// TIA Portal V20 export
FUNCTION "PLC数据交换" : Void   // FC1, LAD
{ S7_Optimized_Access := 'TRUE' }
// stored: SetENOAutomatically false
BEGIN

REGION Network 1
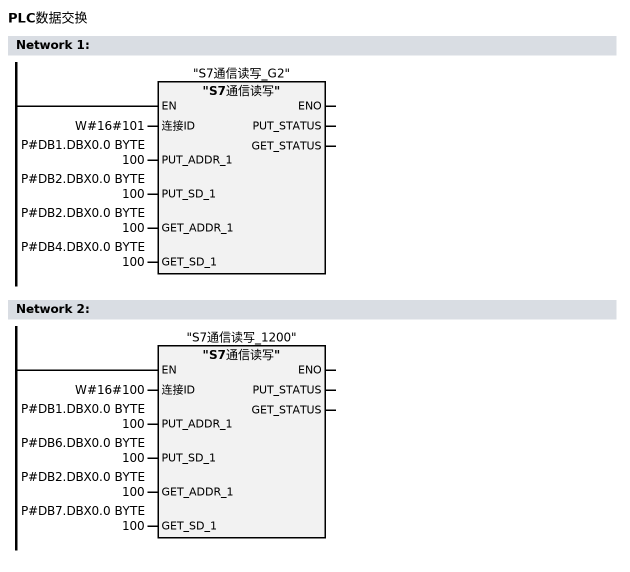
   RUNG wire#powerrail
      "S7通信读写_G2"(连接ID := W#16#101, PUT_ADDR_1 := P#DB1.DBX0.0 BYTE 100, PUT_SD_1 := P#DB2.DBX0.0 BYTE 100, GET_ADDR_1 := P#DB2.DBX0.0 BYTE 100, GET_SD_1 := P#DB4.DBX0.0 BYTE 100, PUT_STATUS =>, GET_STATUS =>)
   END_RUNG
   // the same network as SCL:
   "S7通信读写_G2"(连接ID := W#16#101,   // "S7通信读写"
               PUT_ADDR_1 := P#DB1.DBX0.0 BYTE 100,
               PUT_SD_1 := P#DB2.DBX0.0 BYTE 100,
               GET_ADDR_1 := P#DB2.DBX0.0 BYTE 100,
               GET_SD_1 := P#DB4.DBX0.0 BYTE 100);
END_REGION

REGION Network 2
   RUNG wire#powerrail
      "S7通信读写_1200"(连接ID := W#16#100, PUT_ADDR_1 := P#DB1.DBX0.0 BYTE 100, PUT_SD_1 := P#DB6.DBX0.0 BYTE 100, GET_ADDR_1 := P#DB2.DBX0.0 BYTE 100, GET_SD_1 := P#DB7.DBX0.0 BYTE 100, PUT_STATUS =>, GET_STATUS =>)
   END_RUNG
   // the same network as SCL:
   "S7通信读写_1200"(连接ID := W#16#100,   // "S7通信读写"
                 PUT_ADDR_1 := P#DB1.DBX0.0 BYTE 100,
                 PUT_SD_1 := P#DB6.DBX0.0 BYTE 100,
                 GET_ADDR_1 := P#DB2.DBX0.0 BYTE 100,
                 GET_SD_1 := P#DB7.DBX0.0 BYTE 100);
END_REGION
END_FUNCTION
